TYPE ST_Ramp_Generator :
STRUCT
	tRefreshRate									: LREAL;
	fVelPos											: LREAL	:= 20;
	fVelNeg											: LREAL	:= 40;
END_STRUCT
END_TYPE

(* stored: Version 1.1.0.1
   DUT ST_Ramp_Generator: Id {25d4310d-9aca-49f1-844e-fcbc0fc8628f} *)
